// TwinCAT 3 PLC project snappy
// Title: snappy
// Company: TcHaxx
// Author: densogiaichned
// ProjectVersion: 0.4.0.0
// Description: A Snapshot Testing framework for TwinCAT 3
// ProgramVersion: 3.1.4026.23
// CompilerDefines: TCUNIT
// libraries:
//   rplc, * (TcHaxx)
//   Tc2_Standard, * (Beckhoff Automation GmbH)
//   Tc2_System, * (Beckhoff Automation GmbH)
//   Tc3_JsonXml, * (Beckhoff Automation GmbH)
//   Tc3_Module, * (Beckhoff Automation GmbH)
//   TcUnit, * (www.tcunit.org)
// project tree:
//   DUTs/ E_HESULT_AdsErr.TcTLEO, E_SnappyVerificationState.TcTLEO, ST_VerificationResult.TcDUT, T_SnappyVerifyPort.TcDUT, T_VerifyContent.TcDUT
//   GVLs/ Param_TcHaxx_Snappy.TcGVL
//   ITFs/ I_RpcProxy.TcIO, I_Serializer.TcIO, I_SnappyConfig.TcIO, I_SnappySetup.TcIO, I_SnappySetupConfigSerializer.TcIO, I_SnappySetupConfigBuild.TcIO, I_SnappySetupConfigTestFrameWork.TcIO, I_SnappySetupDefaultsOrRpc.TcIO, I_SnappyVerify.TcIO, I_TestFrameWorkAdapter.TcIO
//   / PlcTask.TcTTO, PlcTaskUnitTest.TcTTO
//   POUs/Adapter/ FB_TcUnitAdapter.TcPOU
//   POUs/ FB_Snappy.TcPOU, MAIN.TcPOU
//   POUs/Helper/ FAILED_AND_NOT_PENDING.TcPOU, PENDING.TcPOU, SUCCEEDED_AND_NOT_PENDING.TcPOU
//   POUs/internal/Config/ FB_SnappyConfig.TcPOU, FB_TestSuiteNameProvider.TcPOU
//   POUs/internal/RPC/ FB_RpcProxy.TcPOU
//   POUs/internal/Serializer/ FB_JsonSerializer.TcPOU
//   TESTs/ PRG_UnitTests.TcPOU
//   TESTs/Serializer/ FB_JsonSerializer_Tests.TcPOU
//   TESTs/snappy/ FB_Snappy_Tests.TcPOU
//   Version/ Global_Version.TcGVL
// real-time tasks:
//   TASK PlcTask: cycle T#10ms, priority 20, ADS port 350
//   TASK PlcTaskUnitTest: cycle T#10ms, priority 1, ADS port 351
//   TASK PlcTaskExamples: cycle T#10ms, priority 21, ADS port 352

CONFIGURATION snappy
    RESOURCE PLC ON TwinCAT3
        TASK PlcTask(INTERVAL := T#10ms, PRIORITY := 20);
        TASK PlcTaskUnitTest(INTERVAL := T#10ms, PRIORITY := 1);
        PROGRAM MAIN WITH PlcTask : MAIN;
        PROGRAM PRG_UnitTests WITH PlcTaskUnitTest : PRG_UnitTests;
    END_RESOURCE
END_CONFIGURATION

// ---- DUTs/E_HESULT_AdsErr.TcTLEO
{attribute 'qualified_only'}
{attribute 'strict'}
TYPE E_HESULT_AdsErr :
(
	ERR_INTERNAL 				:= UDINT_TO_DINT((16#98110000 + 16#1)),		// Internal error.
	ERR_TARGETPORTNOTFOUND 		:= UDINT_TO_DINT((16#98110000 + 16#6)),		// Target port not found – ADS server is not started or is not reachable.
	ERR_TARGETMACHINENOTFOUND 	:= UDINT_TO_DINT((16#98110000 + 16#7)),		// Target computer not found – AMS route was not found. 
	ERR_PORTNOTCONNECTED		:= UDINT_TO_DINT((16#98110000 + 16#D)),		// Port not connected.
	ERR_INVALIDAMSLENGTH		:= UDINT_TO_DINT((16#98110000 + 16#E)),		// Invalid AMS length.
	ERR_INVALIDAMSNETID			:= UDINT_TO_DINT((16#98110000 + 16#F))		// Invalid AMS Net ID.
) DINT;
END_TYPE
//  ERR_INTERNAL = 'UDINT_TO_DINT((16#98110000 + 16#1))'
//  ERR_TARGETPORTNOTFOUND = 'UDINT_TO_DINT((16#98110000 + 16#6))'
//  ERR_TARGETMACHINENOTFOUND = 'UDINT_TO_DINT((16#98110000 + 16#7))'
//  ERR_PORTNOTCONNECTED = 'UDINT_TO_DINT((16#98110000 + 16#D))'
//  ERR_INVALIDAMSLENGTH = 'UDINT_TO_DINT((16#98110000 + 16#E))'
//  ERR_INVALIDAMSNETID = 'UDINT_TO_DINT((16#98110000 + 16#F))'

// ---- DUTs/E_SnappyVerificationState.TcTLEO
{attribute 'qualified_only'}
{attribute 'strict'}
{attribute 'to_string'}
TYPE E_SnappyVerificationState :
(
	eIdle := 0,
	eSend,
	ePending,
	eDone,
	eError := -1
);
END_TYPE
//  eError = '-1'

// ---- DUTs/ST_VerificationResult.TcDUT
{attribute 'no-analysis'}
TYPE ST_VerificationResult :
STRUCT
	hr 		: HRESULT;
	sDiff 	: STRING(Param_TcHaxx_Snappy.cSnappyVerificationResultLength);
END_STRUCT
END_TYPE

// ---- DUTs/T_SnappyVerifyPort.TcDUT
TYPE T_SnappyVerifyPort : UINT (25000..25999); END_TYPE

// ---- DUTs/T_VerifyContent.TcDUT
TYPE T_VerifyContent : STRING(Param_TcHaxx_Snappy.cMaxSizeJsonDocument); END_TYPE

// ---- GVLs/Param_TcHaxx_Snappy.TcGVL
{attribute 'qualified_only'}
{attribute 'no-analysis'}
{attribute 'global_init_slot' := '49992'}
VAR_GLOBAL CONSTANT
	cMaxSizeJsonDocument				: UDINT (16#FF..16#8000) 		:= 16#4000;
	cSnappyVerifyAmsNetID				: T_AmsNetID					:= TcHaxx_rplc.GCL.cLocalAmsNetId;	
	cSnappyVerifyPort					: T_SnappyVerifyPort			:= 25000;
	cSnappyVerifyInstancePath 			: STRING						:= 'TcHaxx.Snappy.Verifier.VerifyService';
	cSnappyVerifySymbol 				: STRING						:= 'Verify';
	cSnappyVerificationResultLength 	: UDINT(16#80..16#4000) 		:= 16#400;	
	cSnappyVerificationTestSuiteLength 	: UDINT(16#80..16#400) 			:= 16#100;
	cSnappyVerificationTestNameLength 	: UDINT(16#80..16#400) 			:= 16#100;			
END_VAR

// ---- Version/Global_Version.TcGVL
{attribute 'TcGenerated'}
{attribute 'no-analysis'}
{attribute 'linkalways'}
// This function has been automatically generated from the project information.
VAR_GLOBAL CONSTANT
	{attribute 'const_non_replaced'}
	stLibVersion_snappy : ST_LibVersion := (iMajor := 0, iMinor := 4, iBuild := 0, iRevision := 0, nFlags := 0, sVersion := '0.4.0.0');
END_VAR

// ---- ITFs/I_RpcProxy.TcIO
INTERFACE I_RpcProxy

PROPERTY bIsConfigured : BOOL
GET
END_GET
END_PROPERTY

METHOD GetVerificationResult : HRESULT

VAR_OUTPUT
	stResult : ST_VerificationResult;
END_VAR
END_METHOD

PROPERTY itfTestFrameWorkAdapter :  I_TestFrameWorkAdapter
GET
END_GET
SET
END_SET
END_PROPERTY

METHOD Verify : HRESULT
VAR_INPUT CONSTANT
	sToVerify	: REFERENCE TO T_VerifyContent;
END_VAR
END_METHOD

END_INTERFACE

// ---- ITFs/I_Serializer.TcIO
INTERFACE I_Serializer

METHOD Serialize : HRESULT
VAR_INPUT
	anyArg	: ANY;
END_VAR
VAR_IN_OUT
	sJsonDocument	: T_VerifyContent;
END_VAR
END_METHOD

END_INTERFACE

// ---- ITFs/I_SnappyConfig.TcIO
INTERFACE I_SnappyConfig EXTENDS I_SnappySetup, I_SnappySetupConfigBuild

PROPERTY bIsConfigured : BOOL
GET
END_GET
END_PROPERTY

PROPERTY itfRpcProxy : I_RpcProxy
GET
END_GET
END_PROPERTY

PROPERTY itfSerializer : I_Serializer
GET
END_GET
END_PROPERTY

PROPERTY itfTestFramework : I_TestFrameWorkAdapter
GET
END_GET
END_PROPERTY

END_INTERFACE

// ---- ITFs/I_SnappySetup.TcIO
INTERFACE I_SnappySetup

METHOD Configure : I_SnappySetupDefaultsOrRpc
VAR_INPUT
END_VAR
END_METHOD

END_INTERFACE

// ---- ITFs/I_SnappySetupConfigSerializer.TcIO
INTERFACE I_SnappySetupConfigSerializer

METHOD UseSerializer : I_SnappySetupConfigBuild
VAR_INPUT
	itfSerializer	: I_Serializer;
END_VAR
END_METHOD

END_INTERFACE

// ---- ITFs/I_SnappySetupConfigBuild.TcIO
INTERFACE I_SnappySetupConfigBuild

METHOD Build : HRESULT
VAR_INPUT
END_VAR
END_METHOD

END_INTERFACE

// ---- ITFs/I_SnappySetupConfigTestFrameWork.TcIO
INTERFACE I_SnappySetupConfigTestFrameWork

METHOD UseTestFramework : I_SnappySetupConfigBuild
VAR_INPUT
	itfTestFramework	: I_TestFrameWorkAdapter;
END_VAR
END_METHOD

METHOD WithoutTestFramework : I_SnappySetupConfigBuild
VAR_INPUT CONSTANT
	sTestSuiteName 	: T_MaxString;
	sTestName		: T_MaxString;
END_VAR
END_METHOD

END_INTERFACE

// ---- ITFs/I_SnappySetupDefaultsOrRpc.TcIO
INTERFACE I_SnappySetupDefaultsOrRpc

METHOD UseDefaults : I_SnappySetupConfigTestFrameWork
VAR_INPUT
END_VAR
END_METHOD

METHOD UseRpcProxy : I_SnappySetupConfigSerializer
VAR_INPUT
	itfRpcProxy	: I_RpcProxy;
END_VAR
END_METHOD

END_INTERFACE

// ---- ITFs/I_SnappyVerify.TcIO
INTERFACE I_SnappyVerify

PROPERTY stVerificationResult : REFERENCE TO ST_VerificationResult
GET
END_GET
END_PROPERTY

METHOD Verify : HRESULT
VAR_INPUT
	anyArg	: ANY;
END_VAR
END_METHOD

END_INTERFACE

// ---- ITFs/I_TestFrameWorkAdapter.TcIO
INTERFACE I_TestFrameWorkAdapter

PROPERTY sTestName : REFERENCE TO T_MaxString
GET
END_GET
END_PROPERTY

PROPERTY sTestSuiteName : REFERENCE TO T_MaxString
GET
END_GET
END_PROPERTY

METHOD Verify : HRESULT
VAR_INPUT
	anyArg	: ANY;
END_VAR
END_METHOD

END_INTERFACE

// ---- POUs/MAIN.TcPOU
PROGRAM INTERNAL MAIN
VAR
END_VAR

END_PROGRAM

// ---- TESTs/PRG_UnitTests.TcPOU
{attribute 'analysis' := '-33'}
PROGRAM INTERNAL PRG_UnitTests
VAR
{IF defined (UNIT_TEST)}	
	fbJsonSerializerTests 	: FB_JsonSerializer_Tests;
	fbSnappyTests			: FB_Snappy_Tests;
{END_IF}
END_VAR

{IF defined (UNIT_TEST)}

TcUnit.RUN();

{END_IF}

END_PROGRAM

// ---- TESTs/Serializer/FB_JsonSerializer_Tests.TcPOU
{attribute 'reflection'}
FUNCTION_BLOCK INTERNAL FINAL FB_JsonSerializer_Tests EXTENDS TcUnit.FB_TestSuite
VAR_INPUT
END_VAR
VAR_OUTPUT
END_VAR
VAR
	{attribute 'instance-path'} 
    {attribute 'noinit'} 
	sTestName			: T_MaxString;
END_VAR

TEST(sTestName);

ShouldSerializeToJsonSuccessfully();

TEST_FINISHED_NAMED(sTestName);

METHOD PRIVATE ShouldSerializeToJsonSuccessfully
VAR_INPUT
END_VAR
VAR_INST
	fbSUT	: FB_JsonSerializer;
	hr		: HRESULT;	
END_VAR

VAR_INST
	stTestData	: ST_AmsAddr;
	sJsonDoc 	: T_VerifyContent;
END_VAR

VAR CONSTANT
	cExpectedJson	: STRING := '{"netId":[1,2,3,4,5,6],"port":1234}';
END_VAR
TEST('ShouldSerializeToJsonSuccessfully');

// Arrange
stTestData.port := 1234;
stTEstData.netId[0]:= 16#1;
stTEstData.netId[1]:= 16#2;
stTEstData.netId[2]:= 16#3;
stTEstData.netId[3]:= 16#4;
stTEstData.netId[4]:= 16#5;
stTEstData.netId[5]:= 16#6;
// Act
hr := fbSUT.Serialize(anyArg:= stTestData, sJsonDocument:= sJsonDoc);
// Assert
AssertEquals_DINT(Expected:= S_OK,
					Actual:= hr,
					Message:= 'Expected HRESULT=S_OK');
AssertEquals_STRING(Expected:= cExpectedJson,
					Actual:= sJsonDoc,
					Message:= 'Expected JSON document $'{"netId":[1,2,3,4,5,6],"port":1234}$'');

TEST_FINISHED();
END_METHOD

END_FUNCTION_BLOCK

// ---- POUs/internal/Serializer/FB_JsonSerializer.TcPOU
{attribute 'no_explicit_call' := 'do not call this POU directly'}
FUNCTION_BLOCK INTERNAL FINAL FB_JsonSerializer IMPLEMENTS I_Serializer
VAR_INPUT
END_VAR
VAR_OUTPUT
END_VAR
VAR
	sDataTypeName 	: STRING;
	fbJsonWriter   	: FB_JsonSaxWriter;
	fbJsonDataType 	: FB_JsonReadWriteDataType;
END_VAR

METHOD Serialize : HRESULT
VAR_INPUT
	anyArg	: ANY;
END_VAR
VAR_IN_OUT
	sJsonDocument	: T_VerifyContent;
END_VAR
VAR
	hr : HRESULT;
END_VAR

IF anyArg.diSize <= 0 OR anyArg.pValue = NULL THEN
	// should never happen...
	Serialize := Tc2_System.E_HRESULTAdsErr.INVALIDPARM;
	RETURN;
END_IF

fbJsonWriter.ResetDocument();
sDataTypeName := fbJsonDataType.GetDatatypeNameByAddress(nData:= TO_UDINT(anyArg.diSize), pData:= anyArg.pValue, hrErrorCode=> hr);
IF FAILED(hr) THEN
	Serialize := hr;
	RETURN;
END_IF
fbJsonDataType.AddJsonValueFromSymbol(fbJsonWriter, sDataTypeName , TO_UDINT(anyArg.diSize), anyArg.pValue, hrErrorCode=> hr);
IF FAILED(hr) THEN
	Serialize := hr;
	RETURN;
END_IF
fbJsonWriter.CopyDocument(sJsonDocument, SIZEOF(sJsonDocument) - 1, hrErrorCode=> hr);
IF FAILED(hr) THEN
	Serialize := hr;
	RETURN;
END_IF

IF sJsonDocument = 'null' AND_THEN SUCCEEDED(hr) THEN
	hr := S_FALSE;
END_IF

Serialize := hr;
END_METHOD

END_FUNCTION_BLOCK

// ---- TESTs/snappy/FB_Snappy_Tests.TcPOU
{attribute 'reflection'}
FUNCTION_BLOCK INTERNAL FINAL FB_Snappy_Tests EXTENDS TcUnit.FB_TestSuite
VAR_INPUT
END_VAR
VAR_OUTPUT
END_VAR
VAR
	{attribute 'instance-path'} 
    {attribute 'noinit'} 
	sTestName			: T_MaxString;
END_VAR

TEST(sTestName);

ShouldInitializeDefaultsSuccessfully();
//Debug();
TEST_FINISHED_NAMED(sTestName);

METHOD PRIVATE Debug
VAR_INST
	
	hr		: HRESULT;		
	fbAdapter : FB_TcUnitAdapter;
END_VAR

TEST('Test some stuff');

// ARRANGE

// ACT and ASSERT
hr := fbAdapter.Verify(anyArg:= _AppInfo);

IF NOT PENDING(hr) THEN
	TEST_FINISHED_NAMED('Test some stuff');
END_IF;
END_METHOD

METHOD PRIVATE ShouldInitializeDefaultsSuccessfully
VAR_INST
	fbSUT		: FB_Snappy;
	hr			: HRESULT;	
END_VAR

TEST('ShuldInitializeDefaultsSuccessfully');

// Arrange
// Act
hr := fbSUT.Configure().UseDefaults().WithoutTestFramework(sTestSuiteName:='MyTestSuite', sTestName:='MyTestName').Build();

// Assert

AssertEquals_DINT(Expected:= S_OK,
				Actual:= hr,
				Message:= 'Expected HRESULT=S_OK');


TEST_FINISHED();
END_METHOD

METHOD PRIVATE Shouldxxx
VAR_INST
	hr		: HRESULT;	
END_VAR

TEST('Shouldxxx');

// Arrange

// Act

// Assert
AssertEquals_DINT(Expected:= S_OK,
					Actual:= hr,
					Message:= 'Expected HRESULT=S_OK');

TEST_FINISHED();
END_METHOD

END_FUNCTION_BLOCK

// ---- POUs/Adapter/FB_TcUnitAdapter.TcPOU
{attribute 'no_explicit_call' := 'do not call this POU directly'}
FUNCTION_BLOCK PUBLIC FINAL FB_TcUnitAdapter IMPLEMENTS I_TestFrameWorkAdapter
VAR
	fbVerify : FB_Snappy;
	eStep : (INIT, VERIFYING, GET_RESULT, FINISHED) := INIT;
END_VAR

PROPERTY sTestName : REFERENCE TO T_MaxString
GET
sTestName REF= GVL_TcUnit.CurrentTestNameBeingCalled;
END_GET
END_PROPERTY

PROPERTY sTestSuiteName : REFERENCE TO T_MaxString
GET
sTestSuiteName REF= GVL_TcUnit.CurrentTestSuiteBeingCalled^.InstancePath;
END_GET
END_PROPERTY

METHOD Verify : HRESULT
VAR_INPUT
	anyArg	: ANY;
END_VAR

VAR	
	hr : HRESULT;
	pTestSuite : POINTER TO FB_TestSuite;
END_VAR
pTestSuite := GVL_TcUnit.CurrentTestSuiteBeingCalled;

IF pTestSuite = NULL THEN
	Verify := Tc2_System.E_HRESULTAdsErr.INVALIDCONTEXT;
	RETURN;
END_IF

CASE eStep OF

	INIT:		
		hr := fbVerify.Configure().UseDefaults().UseTestFramework(THIS^).Build();
		IF SUCCEEDED(hr) THEN
			eStep := VERIFYING;
			hr := S_PENDING;
		ELSE
			pTestSuite^.AssertEquals_DINT(Expected:= S_OK,
								Actual:= hr,
								Message:= 'Configuration failed');			
			eStep := FINISHED;
		END_IF

	VERIFYING:
		hr := fbVerify.Verify(anyArg:= anyArg);
		IF SUCCEEDED_AND_NOT_PENDING(hr)THEN
			eStep := GET_RESULT;
			hr := S_PENDING;
		ELSIF FAILED(hr) AND hr = E_HESULT_AdsErr.ERR_TARGETPORTNOTFOUND THEN
			pTestSuite^.AssertEquals_DINT(Expected:= S_OK,
							Actual:= hr,
							Message:= 'Targetport not found! Make sure, TcHaxx.Snappy.CLI is running, and a ADS route has been established.');
		ELSIF FAILED(hr) THEN
			pTestSuite^.AssertEquals_DINT(Expected:= S_OK,
							Actual:= hr,
							Message:= 'One or more errors occured');
			eStep := FINISHED;
		END_IF

	GET_RESULT:
		hr := fbVerify.stVerificationResult.hr;
		IF FAILED(hr) THEN
				pTestSuite^.AssertEquals_DINT(Expected:= S_OK,
								Actual:= hr,
								Message:= fbVerify.stVerificationResult.sDiff);
		END_IF;
		eStep := FINISHED;

	FINISHED:
		eStep := INIT;
END_CASE

Verify := hr;
END_METHOD

END_FUNCTION_BLOCK

// ---- POUs/FB_Snappy.TcPOU
{attribute 'no_explicit_call' := 'do not call this POU directly'}
FUNCTION_BLOCK FINAL FB_Snappy IMPLEMENTS I_SnappySetup, I_SnappySetupConfigBuild, I_SnappyVerify
VAR_INPUT
END_VAR
VAR_OUTPUT
END_VAR

VAR
//	{attribute 'hide'}
	fbConfig					: FB_SnappyConfig;
	itfConfig					: I_SnappyConfig := fbConfig; 
	fbTestSuiteNameProvider		: FB_TestSuiteNameProvider;
	itfTestFrameWork			: I_TestFrameWorkAdapter := fbTestSuiteNameProvider;
	stVerificationResultField 	: ST_VerificationResult;
END_VAR

{attribute 'estimated-stack-usage' := '4096'}
METHOD Build : HRESULT
Build := itfConfig.Build();

IF FAILED(Build) THEN
	RETURN;
END_IF

IF THIS^.itfConfig.itfTestFramework <> NULL THEN
	THIS^.itfTestFrameWork := THIS^.itfConfig.itfTestFramework;
END_IF
END_METHOD

{attribute 'estimated-stack-usage' := '4096'}
METHOD Configure : I_SnappySetupDefaultsOrRpc
Configure := THIS^.itfConfig.Configure();
END_METHOD

PROPERTY stVerificationResult : REFERENCE TO ST_VerificationResult
GET
stVerificationResult REF= THIS^.stVerificationResultField;
END_GET
END_PROPERTY

METHOD Verify : HRESULT
VAR_INPUT
	anyArg	: ANY;
END_VAR

VAR
	hr 		: HRESULT;
END_VAR


VAR_INST
	sJDoc			: T_VerifyContent;
	eState			: E_SnappyVerificationState;
	hrLastErrorCode : HRESULT;
END_VAR

IF NOT itfConfig.bIsConfigured THEN
	Verify := Tc2_system.E_HRESULTAdsErr.NOTREADY;
	RETURN;
END_IF

CASE eState OF
	
	E_SnappyVerificationState.eIdle:
	itfConfig.itfRpcProxy.itfTestFrameWorkAdapter := THIS^.itfConfig.itfTestFramework;
	hr := itfConfig.itfSerializer.Serialize(anyArg:= anyArg, sJsonDocument:= sJDoc);
	IF FAILED(hr) THEN
		hrLastErrorCode := hr;
		eState := E_SnappyVerificationState.eError;
	ELSE
		hrLastErrorCode := S_PENDING;
		eState := E_SnappyVerificationState.eSend;
	END_IF

	E_SnappyVerificationState.eSend:		
		hr := itfConfig.itfRpcProxy.Verify(sToVerify:= sJDoc);
		IF SUCCEEDED(hr) THEN
			eState := E_SnappyVerificationState.ePending;
		ELSIF FAILED(hr) THEN
			hrLastErrorCode := hr;
			eState := E_SnappyVerificationState.eError;
		END_IF
		
	E_SnappyVerificationState.ePending:
		hr := itfConfig.itfRpcProxy.GetVerificationResult(stResult => stVerificationResultField);
		hrLastErrorCode := hr;
		IF SUCCEEDED_AND_NOT_PENDING(hr) THEN
			eState := E_SnappyVerificationState.eDone;
		ELSIF FAILED(hr) THEN
			eState := E_SnappyVerificationState.eError;
		END_IF

	E_SnappyVerificationState.eDone:
		eState := E_SnappyVerificationState.eIdle;

	E_SnappyVerificationState.eError:
		eState := E_SnappyVerificationState.eIdle;
		
END_CASE

Verify := hrLastErrorCode;
END_METHOD

END_FUNCTION_BLOCK

// ---- POUs/internal/Config/FB_SnappyConfig.TcPOU
{attribute 'no_explicit_call' := 'do not call this POU directly'}
FUNCTION_BLOCK INTERNAL FINAL FB_SnappyConfig IMPLEMENTS I_SnappyConfig, I_SnappySetupDefaultsOrRpc, I_SnappySetupConfigSerializer, I_SnappySetupConfigTestFrameWork
VAR
	eConfigState		: (NOT_CONFIGURED, IS_CONFIGURED) := NOT_CONFIGURED;
END_VAR

VAR
	itfSerializerField		: I_Serializer 	:= NULL;
	itfRpcProxyField		: I_RpcProxy	:= NULL;
	itfTestFrameworkField	: I_TestFrameWorkAdapter := NULL;
END_VAR

VAR
	fbJsonSerializer	: FB_JsonSerializer;
	fbRpcProxy			: FB_RpcProxy;
	fbTestNamesProvider : FB_TestSuiteNameProvider;
END_VAR

PROPERTY bIsConfigured : BOOL
GET
bIsConfigured := eConfigState = IS_CONFIGURED;
END_GET
END_PROPERTY

METHOD Build : HRESULT

IF itfRpcProxyField = NULL THEN
	Build := Tc2_System.E_HRESULTAdsErr.INVALIDPARM;
	RETURN;
END_IF

IF itfSerializerField = NULL THEN
	Build := Tc2_System.E_HRESULTAdsErr.INVALIDPARM;
	RETURN;
END_IF

eConfigState := IS_CONFIGURED;
END_METHOD

METHOD Configure : I_SnappySetupDefaultsOrRpc
Configure := THIS^;
IF bIsConfigured THEN
	RETURN;
END_IF
END_METHOD

PROPERTY itfRpcProxy : I_RpcProxy
GET
itfRpcProxy := itfRpcProxyField;
END_GET
END_PROPERTY

PROPERTY itfSerializer : I_Serializer
GET
itfSerializer := itfSerializerField;
END_GET
END_PROPERTY

PROPERTY itfTestFramework : I_TestFrameWorkAdapter
GET
itfTestFramework := itfTestFrameworkField;
END_GET
END_PROPERTY

METHOD UseDefaults : I_SnappySetupConfigTestFrameWork
UseDefaults := THIS^;

IF bIsConfigured THEN
	RETURN;
END_IF

THIS^.itfSerializerField 	:= fbJsonSerializer;
THIS^.itfRpcProxyField 		:= fbRpcProxy;
END_METHOD

METHOD UseRpcProxy : I_SnappySetupConfigSerializer
VAR_INPUT
	itfRpcProxy	: I_RpcProxy;
END_VAR
UseRpcProxy := THIS^;

IF bIsConfigured THEN
	RETURN;
END_IF

THIS^.itfRpcProxyField := itfRpcProxy;
END_METHOD

METHOD UseSerializer : I_SnappySetupConfigBuild
VAR_INPUT
	itfSerializer	: I_Serializer;
END_VAR
UseSerializer := THIS^;

IF bIsConfigured THEN
	RETURN;
END_IF

THIS^.itfSerializerField := itfSerializer;
END_METHOD

METHOD UseTestFramework : I_SnappySetupConfigBuild
VAR_INPUT
	itfTestFramework	: I_TestFrameWorkAdapter;
END_VAR
UseTestFramework := THIS^;

IF bIsConfigured THEN
	RETURN;
END_IF

THIS^.itfTestFrameworkField := itfTestFramework;
END_METHOD

METHOD WithoutTestFramework : I_SnappySetupConfigBuild
VAR_INPUT CONSTANT
	sTestSuiteName 	: T_MaxString;
	sTestName		: T_MaxString;
END_VAR
WithoutTestFramework := THIS^;

THIS^.fbTestNamesProvider.SetTestNames(sTestSuiteName, sTestName);
THIS^.itfTestFrameworkField := THIS^.fbTestNamesProvider;

IF bIsConfigured THEN
	RETURN;
END_IF
END_METHOD

END_FUNCTION_BLOCK

// ---- POUs/internal/RPC/FB_RpcProxy.TcPOU
{attribute 'no_explicit_call' := 'do not call this POU directly'}
FUNCTION_BLOCK INTERNAL FB_RpcProxy IMPLEMENTS I_RpcProxy
VAR_INPUT
END_VAR
VAR_OUTPUT
END_VAR
VAR
	fbRpcSnappyVerify		: FB_RPC_Dynamic;
	sAmsNetID				: T_AmsNetID 			:= Param_TcHaxx_Snappy.cSnappyVerifyAmsNetID;
	nAmsPort				: T_AmsPort				:= Param_TcHaxx_Snappy.cSnappyVerifyPort;
	sInstancePathLocalField	: STRING				:= Param_TcHaxx_Snappy.cSnappyVerifyInstancePath;
	sSymbolLocalField		: STRING				:= Param_TcHaxx_Snappy.cSnappyVerifySymbol;
	bIsConfiguredField		: BOOL					:= FALSE;
	stVerificationResult	: ST_VerificationResult;
	itfTestFrameWorkField	: I_TestFrameWorkAdapter;
END_VAR

PROPERTY bIsConfigured : BOOL
GET
bIsConfigured := bIsConfiguredField;
END_GET
END_PROPERTY

METHOD GetVerificationResult : HRESULT
VAR_OUTPUT
	stResult : ST_VerificationResult;
END_VAR

VAR
	stAdsStatus	: TcHaxx_rplc.ST_AdsStatus;
END_VAR
GetVerificationResult := S_PENDING;

stAdsStatus := THIS^.fbRpcSnappyVerify.Invoke();

IF NOT stAdsStatus.bBusy AND NOT stAdsStatus.bError THEN
	GetVerificationResult := S_OK;
	stResult := stVerificationResult;
	RETURN;
ELSIF stAdsStatus.bError THEN
	GetVerificationResult := TO_DINT(stAdsStatus.nError);
	IF GetVerificationResult > 0 THEN
		GetVerificationResult := TO_DINT(TO_UDINT(GetVerificationResult) OR 16#98110000);
	END_IF
	RETURN;
END_IF
END_METHOD

PROPERTY itfTestFrameWorkAdapter : I_TestFrameWorkAdapter
GET
itfTestFrameWorkAdapter := THIS^.itfTestFrameWorkField;
END_GET
SET
THIS^.itfTestFrameWorkField := itfTestFrameWorkAdapter;
END_SET
END_PROPERTY

METHOD Verify : HRESULT
VAR_INPUT CONSTANT
	sToVerify			: REFERENCE TO T_VerifyContent;
END_VAR
VAR
	hr			: HRESULT;
	stAdsStatus	: TcHaxx_rplc.ST_AdsStatus;
	
	
	sTestSuiteName : STRING(Param_TcHaxx_Snappy.cSnappyVerificationTestSuiteLength) := 'ATestSuiteName';
	sTestName : STRING(Param_TcHaxx_Snappy.cSnappyVerificationTestNameLength) := 'ATestName';
END_VAR
IF NOT bIsConfiguredField THEN
	hr := fbRpcSnappyVerify.Configure()
			.WithAmsNetId(sAmsNetId:= THIS^.sAmsNetID)
			.WithAmsPort(nAmsPort:= THIS^.nAmsPort)
			.WithSymbolPath(sInstancePath:= THIS^.sInstancePathLocalField, sSymbol:= THIS^.sSymbolLocalField)
			.Build();
	bIsConfiguredField := SUCCEEDED(hr);
END_IF;

IF NOT bIsConfigured THEN
	Verify := E_HRESULTAdsErr.NOTINIT;
	RETURN;
END_IF

IF itfTestFrameWorkField <> NULL THEN
	sTestSuiteName 	:= itfTestFrameWorkField.sTestSuiteName;
	sTestName 		:= itfTestFrameWorkField.sTestName;
END_IF

stAdsStatus := fbRpcSnappyVerify.VarInput(anyArg:= sTestSuiteName)
								.VarInput(anyArg:= sTestName)
							 	.VarInput(anyArg:= sToVerify)
								.ReturnValue(anyRetVal:= stVerificationResult)
								.Invoke();
IF stAdsStatus.bError THEN
	Verify := TO_DINT(stAdsStatus.nError);
	RETURN;
END_IF

Verify := S_PENDING;
END_METHOD

END_FUNCTION_BLOCK

// ---- POUs/internal/Config/FB_TestSuiteNameProvider.TcPOU
{attribute 'no_explicit_call' := 'do not call this POU directly'}
FUNCTION_BLOCK INTERNAL FINAL FB_TestSuiteNameProvider IMPLEMENTS I_TestFrameWorkAdapter
VAR_INPUT
END_VAR
VAR_OUTPUT
END_VAR
VAR
	sTestSuiteNameField 	: T_MaxString;
	sTestNameField			: T_MaxString;
END_VAR

METHOD INTERNAL SetTestNames
VAR_INPUT CONSTANT
	sTestSuiteName 	: REFERENCE TO T_MaxString;
	sTestName		: REFERENCE TO T_MaxString;
END_VAR

sTestSuiteNameField := sTestSuiteName;
sTestNameField := sTestName;
END_METHOD

PROPERTY sTestName : REFERENCE TO Tc2_System.T_MaxString
GET
sTestName REF= sTestNameField;
END_GET
END_PROPERTY

PROPERTY sTestSuiteName : REFERENCE TO Tc2_System.T_MaxString
GET
sTestSuiteName REF= sTestSuiteNameField;
END_GET
END_PROPERTY

METHOD Verify : HRESULT
VAR_INPUT
	{attribute 'analysis' := '-33'}
	anyArg	: __SYSTEM.AnyType;
END_VAR
Verify := Tc2_System.E_HRESULTAdsErr.ACCESSDENIED;
END_METHOD

END_FUNCTION_BLOCK

// ---- POUs/Helper/SUCCEEDED_AND_NOT_PENDING.TcPOU
FUNCTION SUCCEEDED_AND_NOT_PENDING : BOOL
VAR_INPUT
	hr 	: DINT;
END_VAR
VAR
END_VAR

SUCCEEDED_AND_NOT_PENDING := hr >= 0 AND hr <> S_PENDING;

END_FUNCTION

// ---- POUs/Helper/PENDING.TcPOU
FUNCTION PENDING : BOOL
VAR_INPUT
	hr 	: DINT;
END_VAR
VAR
END_VAR

PENDING := hr = S_PENDING;

END_FUNCTION

// ---- POUs/Helper/FAILED_AND_NOT_PENDING.TcPOU
FUNCTION FAILED_AND_NOT_PENDING : BOOL
VAR_INPUT
	hr 	: DINT;
END_VAR
VAR
END_VAR

FAILED_AND_NOT_PENDING := hr <> S_OK AND hr <> S_PENDING;

END_FUNCTION
